PROGRAM PTM1
VAR
END_VAR

END_PROGRAM

(* stored: Version 1.1.0.1, ProductVersion 3.1.4022.3
   POU PTM1: Id {a6d69970-ba4c-4978-992b-8d62b2a83208}, SpecialFunc None *)
